// TIA Portal V20 export
TYPE "sAxis_SS"
   STRUCT
      bHome : Bool;   // 原点传感器
      bFW : Bool := TRUE;   // 前限位
      bBW : Bool := TRUE;   // 后限位
   END_STRUCT;
END_TYPE
